# EPICS substitutions: iocBoot/iocnamWin/substitutions/canberra_13.substitutions
file "$(MCA)/mcaApp/Db/simple_mca.db"
{
pattern
{P           M       DTYP           INP         PREC  CHANS}
{namWin:med:   mca1  "asynMCA"   "@asyn(AIM2/1 0)"    3  2048}
{namWin:med:   mca2  "asynMCA"   "@asyn(AIM2/1 1)"    3  2048}
{namWin:med:   mca3  "asynMCA"   "@asyn(AIM2/1 2)"    3  2048}
{namWin:med:   mca4  "asynMCA"   "@asyn(AIM2/2 0)"    3  2048}
{namWin:med:   mca5  "asynMCA"   "@asyn(AIM2/2 1)"    3  2048}
{namWin:med:   mca6  "asynMCA"   "@asyn(AIM2/2 2)"    3  2048}
{namWin:med:   mca7  "asynMCA"   "@asyn(AIM3/1 0)"    3  2048}
{namWin:med:   mca8  "asynMCA"   "@asyn(AIM3/1 1)"    3  2048}
{namWin:med:   mca9  "asynMCA"   "@asyn(AIM3/1 2)"    3  2048}
{namWin:med:   mca10 "asynMCA"   "@asyn(AIM3/2 0)"    3  2048}
{namWin:med:   mca11 "asynMCA"   "@asyn(AIM3/3 1)"    3  2048}
{namWin:med:   mca12 "asynMCA"   "@asyn(AIM3/4 2)"    3  2048}
{namWin:med:   mca13 "asynMCA"   "@asyn(AIM3/2 3)"    3  2048}
{namWin:med:   mca0  "Soft Channel"   ""     3  2048}
}

file "$(MCA)/mcaApp/Db/icb_amp.db"
{
pattern
{P			AMP		PORT}
{namWin:med:	amp1	"icbAmp1"}
{namWin:med:	amp2	"icbAmp2"}
{namWin:med:	amp3	"icbAmp3"}
{namWin:med:	amp4	"icbAmp4"}
{namWin:med:	amp5	"icbAmp5"}
{namWin:med:	amp6	"icbAmp6"}
{namWin:med:	amp7	"icbAmp7"}
{namWin:med:	amp8	"icbAmp8"}
{namWin:med:	amp9	"icbAmp9"}
{namWin:med:	amp10	"icbAmp10"}
{namWin:med:	amp11	"icbAmp11"}
{namWin:med:	amp12	"icbAmp12"}
{namWin:med:	amp13	"icbAmp13"}
}

file "$(MCA)/mcaApp/Db/icb_adc.db"
{
pattern
{P			ADC		PORT}
{namWin:med:	adc1	"icbAdc1"}
{namWin:med:	adc2	"icbAdc2"}
{namWin:med:	adc3	"icbAdc3"}
{namWin:med:	adc4	"icbAdc4"}
}

file "$(MCA)/mcaApp/Db/icb_hvps.db"
{
pattern
{P			HVPS	LIMIT	PORT}
{namWin:med:	hvps1	1000	"icbHvps1"}
}
